% RSLogix 500 project MULTI_POSITION_SERVO.RSS, saved by version 8.30.00.16 %
PROJECT "UNTITLED"    % processor: Bul.1763 MicroLogix 1100 Series B %

PROGRAM FILES
  LAD 2 "MAIN"  4 rungs
  LAD 3 "I/O"  8 rungs
  LAD 4 "CONTROLS"  22 rungs

DATA FILES
  O0 OUTPUT  5 elements
  I1 INPUT  7 elements
  S2 STATUS  66 elements
  B3 BINARY  3 elements
  T4 TIMER  3 elements
  C5 COUNTER  1 elements
  R6 CONTROL  1 elements
  N7 INTEGER  2 elements
  F8 FLOAT  1 elements

LADDER 2 "MAIN"
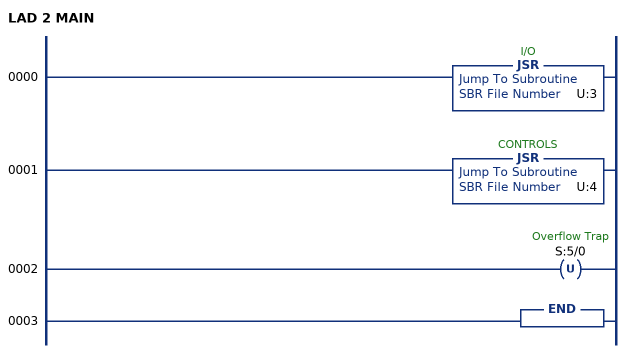
% Rung: 0 %
SOR JSR U:3 EOR
%   U:3  "I/O" %
% Rung: 1 %
SOR JSR U:4 EOR
%   U:4  "CONTROLS" %
% Rung: 2 %
SOR OTU S:5/0 EOR
%   S:5/0  "Overflow Trap" %
% Rung: 3 %
SOR END EOR

LADDER 3 "I/O"
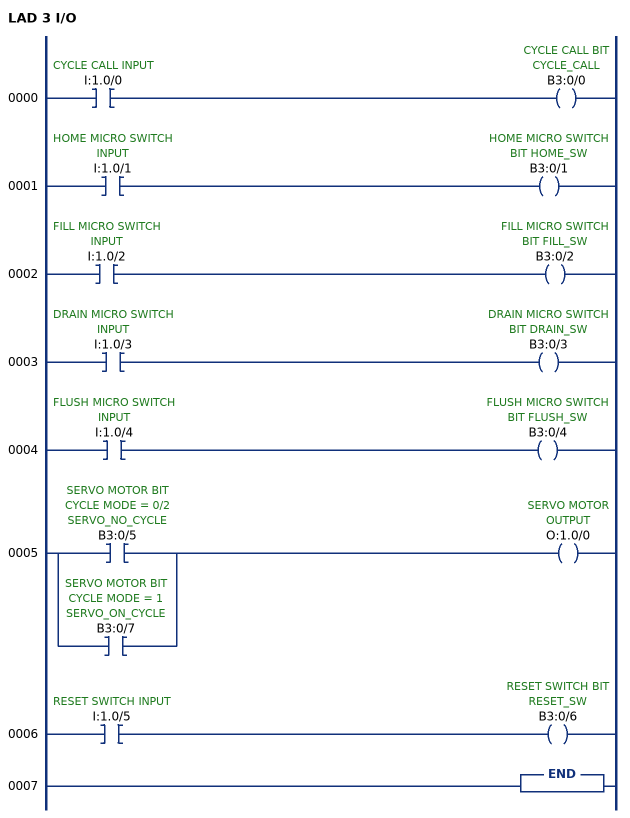
% Rung: 0 %
SOR XIC I:1.0/0 OTE B3:0/0 EOR
%   I:1.0/0  "CYCLE CALL INPUT" %
%   B3:0/0  CYCLE_CALL  "CYCLE CALL BIT" %
% Rung: 1 %
SOR XIC I:1.0/1 OTE B3:0/1 EOR
%   I:1.0/1  "HOME MICRO SWITCH INPUT" %
%   B3:0/1  HOME_SW  "HOME MICRO SWITCH BIT" %
% Rung: 2 %
SOR XIC I:1.0/2 OTE B3:0/2 EOR
%   I:1.0/2  "FILL MICRO SWITCH INPUT" %
%   B3:0/2  FILL_SW  "FILL MICRO SWITCH BIT" %
% Rung: 3 %
SOR XIC I:1.0/3 OTE B3:0/3 EOR
%   I:1.0/3  "DRAIN MICRO SWITCH INPUT" %
%   B3:0/3  DRAIN_SW  "DRAIN MICRO SWITCH BIT" %
% Rung: 4 %
SOR XIC I:1.0/4 OTE B3:0/4 EOR
%   I:1.0/4  "FLUSH MICRO SWITCH INPUT" %
%   B3:0/4  FLUSH_SW  "FLUSH MICRO SWITCH BIT" %
% Rung: 5 %
SOR BST XIC B3:0/5 NXB XIC B3:0/7 BND OTE O:1.0/0 EOR
%   B3:0/5  SERVO_NO_CYCLE  "SERVO MOTOR BIT CYCLE MODE = 0/2" %
%   B3:0/7  SERVO_ON_CYCLE  "SERVO MOTOR BIT CYCLE MODE = 1" %
%   O:1.0/0  "SERVO MOTOR OUTPUT" %
% Rung: 6 %
SOR XIC I:1.0/5 OTE B3:0/6 EOR
%   I:1.0/5  "RESET SWITCH INPUT" %
%   B3:0/6  RESET_SW  "RESET SWITCH BIT" %
% Rung: 7 %
SOR END EOR

LADDER 4 "CONTROLS"
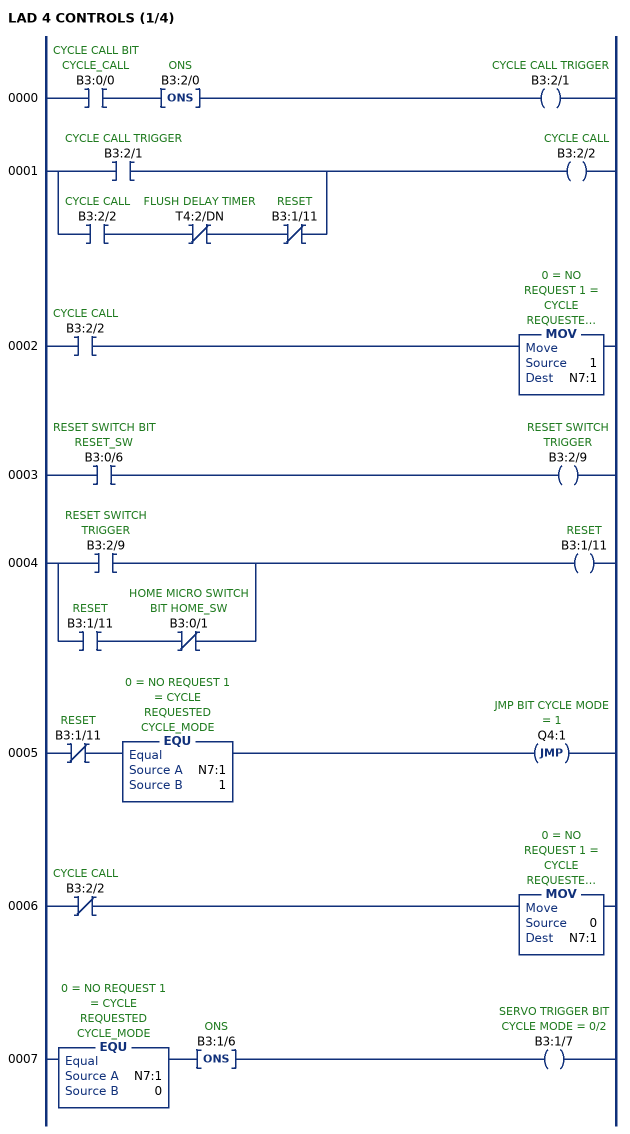
% Rung: 0 %
SOR XIC B3:0/0 ONS B3:2/0 OTE B3:2/1 EOR
%   B3:0/0  CYCLE_CALL  "CYCLE CALL BIT" %
%   B3:2/0  "ONS" %
%   B3:2/1  "CYCLE CALL TRIGGER" %
% Rung: 1 %
SOR BST XIC B3:2/1 NXB XIC B3:2/2 XIO T4:2/DN XIO B3:1/11 BND OTE B3:2/2 EOR
%   B3:2/1  "CYCLE CALL TRIGGER" %
%   B3:2/2  "CYCLE CALL" %
%   T4:2/DN  "FLUSH DELAY TIMER" %
%   B3:1/11  "RESET" %
% Rung: 2 %
SOR XIC B3:2/2 MOV 1 N7:1 EOR
%   B3:2/2  "CYCLE CALL" %
%   N7:1  CYCLE_MODE  "0 = NO REQUEST 1 = CYCLE REQUESTED" %
% Rung: 3 %
SOR XIC B3:0/6 OTE B3:2/9 EOR
%   B3:0/6  RESET_SW  "RESET SWITCH BIT" %
%   B3:2/9  "RESET SWITCH TRIGGER" %
% Rung: 4 %
SOR BST XIC B3:2/9 NXB XIC B3:1/11 XIO B3:0/1 BND OTE B3:1/11 EOR
%   B3:2/9  "RESET SWITCH TRIGGER" %
%   B3:1/11  "RESET" %
%   B3:0/1  HOME_SW  "HOME MICRO SWITCH BIT" %
% Rung: 5 %
SOR XIO B3:1/11 EQU N7:1 1 JMP Q4:1 EOR
%   B3:1/11  "RESET" %
%   N7:1  CYCLE_MODE  "0 = NO REQUEST 1 = CYCLE REQUESTED" %
%   Q4:1  "JMP BIT CYCLE MODE = 1" %
% Rung: 6 %
SOR XIO B3:2/2 MOV 0 N7:1 EOR
%   B3:2/2  "CYCLE CALL" %
%   N7:1  CYCLE_MODE  "0 = NO REQUEST 1 = CYCLE REQUESTED" %
% Rung: 7 %
SOR EQU N7:1 0 ONS B3:1/6 OTE B3:1/7 EOR
%   N7:1  CYCLE_MODE  "0 = NO REQUEST 1 = CYCLE REQUESTED" %
%   B3:1/6  "ONS" %
%   B3:1/7  "SERVO TRIGGER BIT CYCLE MODE = 0/2" %

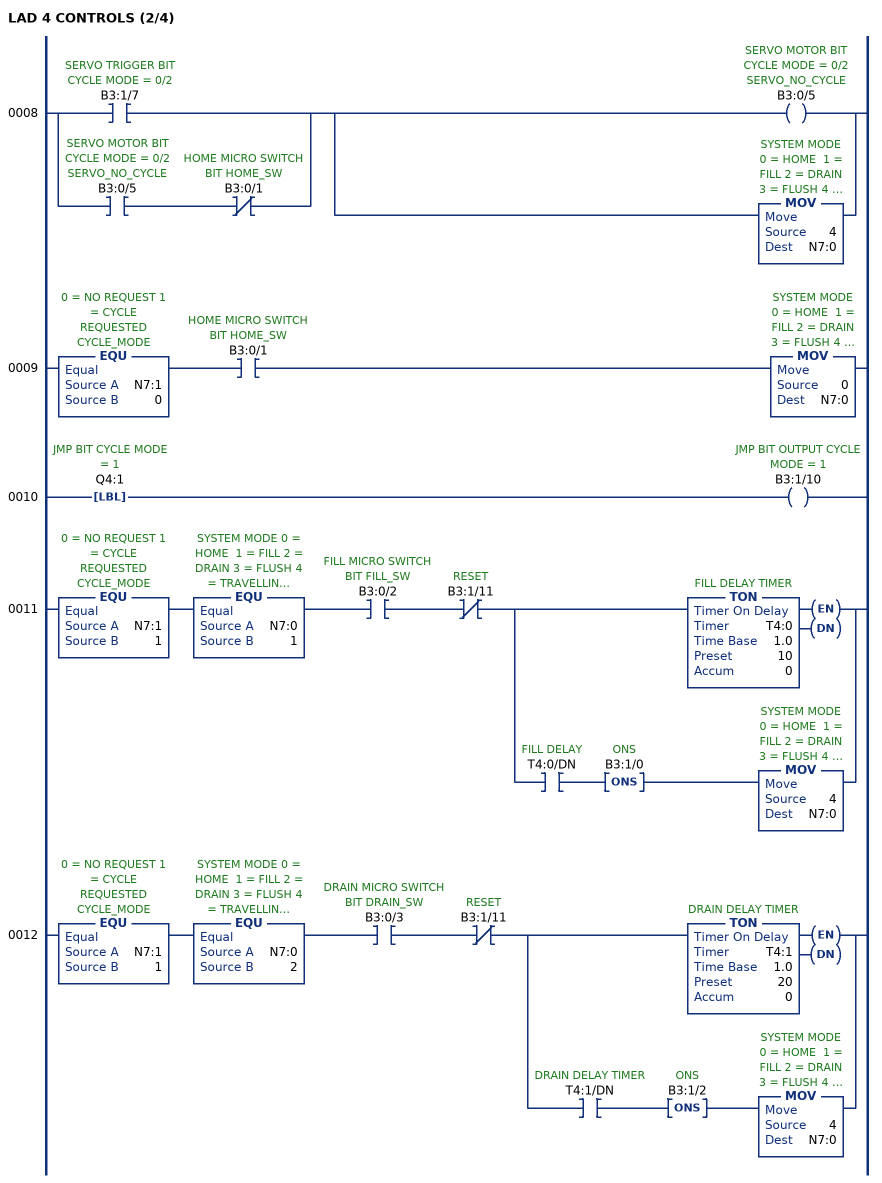
% Rung: 8 %
SOR BST XIC B3:1/7 NXB XIC B3:0/5 XIO B3:0/1 BND BST OTE B3:0/5 NXB MOV 4 N7:0 BND EOR
%   B3:1/7  "SERVO TRIGGER BIT CYCLE MODE = 0/2" %
%   B3:0/5  SERVO_NO_CYCLE  "SERVO MOTOR BIT CYCLE MODE = 0/2" %
%   B3:0/1  HOME_SW  "HOME MICRO SWITCH BIT" %
%   N7:0  SYSTEM_MODE  "SYSTEM MODE 0 = HOME  1 = FILL 2 = DRAIN 3 = FLUSH 4 = TRAVELLING" %
% Rung: 9 %
SOR EQU N7:1 0 XIC B3:0/1 MOV 0 N7:0 EOR
%   N7:1  CYCLE_MODE  "0 = NO REQUEST 1 = CYCLE REQUESTED" %
%   B3:0/1  HOME_SW  "HOME MICRO SWITCH BIT" %
%   N7:0  SYSTEM_MODE  "SYSTEM MODE 0 = HOME  1 = FILL 2 = DRAIN 3 = FLUSH 4 = TRAVELLING" %
% Rung: 10 %
SOR LBL Q4:1 OTE B3:1/10 EOR
%   Q4:1  "JMP BIT CYCLE MODE = 1" %
%   B3:1/10  "JMP BIT OUTPUT CYCLE MODE = 1" %
% Rung: 11 %
SOR EQU N7:1 1 EQU N7:0 1 XIC B3:0/2 XIO B3:1/11 BST TON T4:0 1.0 10 0 NXB XIC T4:0/DN ONS B3:1/0 MOV 4 N7:0 BND EOR
%   N7:1  CYCLE_MODE  "0 = NO REQUEST 1 = CYCLE REQUESTED" %
%   N7:0  SYSTEM_MODE  "SYSTEM MODE 0 = HOME  1 = FILL 2 = DRAIN 3 = FLUSH 4 = TRAVELLING" %
%   B3:0/2  FILL_SW  "FILL MICRO SWITCH BIT" %
%   B3:1/11  "RESET" %
%   T4:0  "FILL DELAY TIMER" %
%   T4:0/DN  "FILL DELAY" %
%   B3:1/0  "ONS" %
% Rung: 12 %
SOR EQU N7:1 1 EQU N7:0 2 XIC B3:0/3 XIO B3:1/11 BST TON T4:1 1.0 20 0 NXB XIC T4:1/DN ONS B3:1/2 MOV 4 N7:0 BND EOR
%   N7:1  CYCLE_MODE  "0 = NO REQUEST 1 = CYCLE REQUESTED" %
%   N7:0  SYSTEM_MODE  "SYSTEM MODE 0 = HOME  1 = FILL 2 = DRAIN 3 = FLUSH 4 = TRAVELLING" %
%   B3:0/3  DRAIN_SW  "DRAIN MICRO SWITCH BIT" %
%   B3:1/11  "RESET" %
%   T4:1  "DRAIN DELAY TIMER" %
%   T4:1/DN  "DRAIN DELAY TIMER" %
%   B3:1/2  "ONS" %

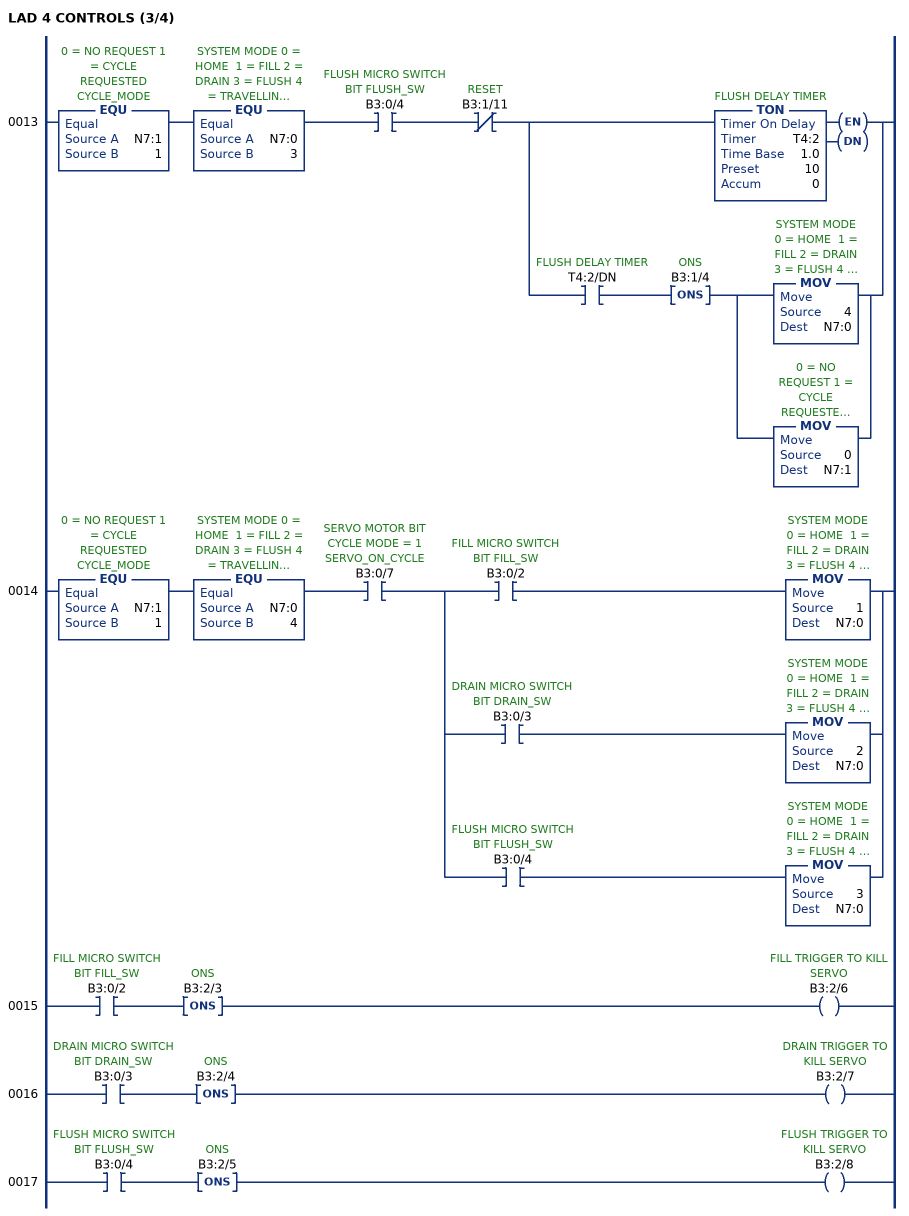
% Rung: 13 %
SOR EQU N7:1 1 EQU N7:0 3 XIC B3:0/4 XIO B3:1/11 BST TON T4:2 1.0 10 0 NXB XIC T4:2/DN ONS B3:1/4 BST MOV 4 N7:0 NXB MOV 0 N7:1 BND BND EOR
%   N7:1  CYCLE_MODE  "0 = NO REQUEST 1 = CYCLE REQUESTED" %
%   N7:0  SYSTEM_MODE  "SYSTEM MODE 0 = HOME  1 = FILL 2 = DRAIN 3 = FLUSH 4 = TRAVELLING" %
%   B3:0/4  FLUSH_SW  "FLUSH MICRO SWITCH BIT" %
%   B3:1/11  "RESET" %
%   T4:2  "FLUSH DELAY TIMER" %
%   T4:2/DN  "FLUSH DELAY TIMER" %
%   B3:1/4  "ONS" %
% Rung: 14 %
SOR EQU N7:1 1 EQU N7:0 4 XIC B3:0/7 BST XIC B3:0/2 MOV 1 N7:0 NXB XIC B3:0/3 MOV 2 N7:0 NXB XIC B3:0/4 MOV 3 N7:0 BND EOR
%   N7:1  CYCLE_MODE  "0 = NO REQUEST 1 = CYCLE REQUESTED" %
%   N7:0  SYSTEM_MODE  "SYSTEM MODE 0 = HOME  1 = FILL 2 = DRAIN 3 = FLUSH 4 = TRAVELLING" %
%   B3:0/7  SERVO_ON_CYCLE  "SERVO MOTOR BIT CYCLE MODE = 1" %
%   B3:0/2  FILL_SW  "FILL MICRO SWITCH BIT" %
%   B3:0/3  DRAIN_SW  "DRAIN MICRO SWITCH BIT" %
%   B3:0/4  FLUSH_SW  "FLUSH MICRO SWITCH BIT" %
% Rung: 15 %
SOR XIC B3:0/2 ONS B3:2/3 OTE B3:2/6 EOR
%   B3:0/2  FILL_SW  "FILL MICRO SWITCH BIT" %
%   B3:2/3  "ONS" %
%   B3:2/6  "FILL TRIGGER TO KILL SERVO" %
% Rung: 16 %
SOR XIC B3:0/3 ONS B3:2/4 OTE B3:2/7 EOR
%   B3:0/3  DRAIN_SW  "DRAIN MICRO SWITCH BIT" %
%   B3:2/4  "ONS" %
%   B3:2/7  "DRAIN TRIGGER TO KILL SERVO" %
% Rung: 17 %
SOR XIC B3:0/4 ONS B3:2/5 OTE B3:2/8 EOR
%   B3:0/4  FLUSH_SW  "FLUSH MICRO SWITCH BIT" %
%   B3:2/5  "ONS" %
%   B3:2/8  "FLUSH TRIGGER TO KILL SERVO" %

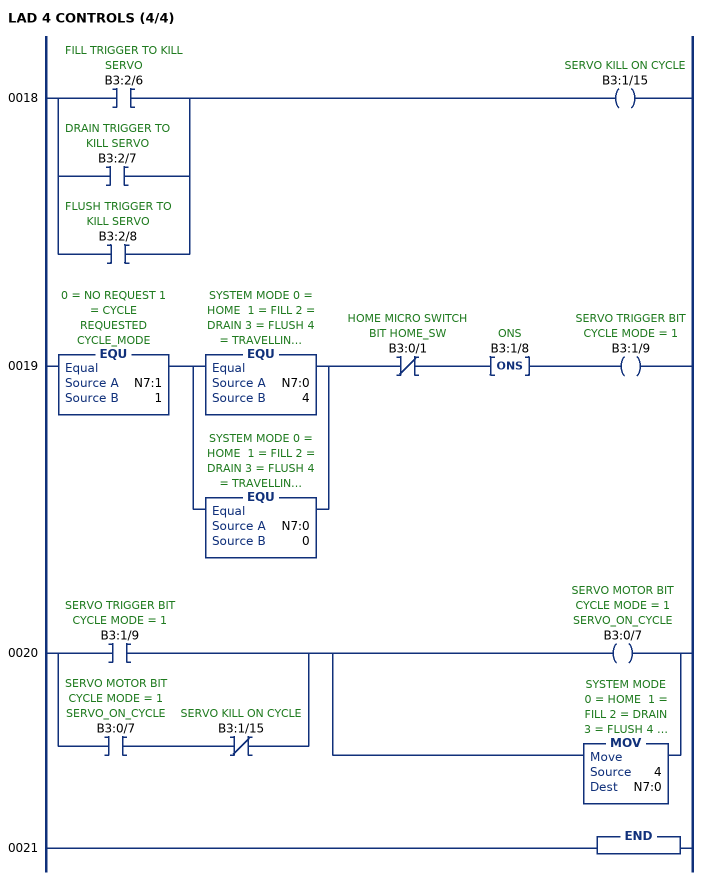
% Rung: 18 %
SOR BST XIC B3:2/6 NXB XIC B3:2/7 NXB XIC B3:2/8 BND OTE B3:1/15 EOR
%   B3:2/6  "FILL TRIGGER TO KILL SERVO" %
%   B3:2/7  "DRAIN TRIGGER TO KILL SERVO" %
%   B3:2/8  "FLUSH TRIGGER TO KILL SERVO" %
%   B3:1/15  "SERVO KILL ON CYCLE" %
% Rung: 19 %
SOR EQU N7:1 1 BST EQU N7:0 4 NXB EQU N7:0 0 BND XIO B3:0/1 ONS B3:1/8 OTE B3:1/9 EOR
%   N7:1  CYCLE_MODE  "0 = NO REQUEST 1 = CYCLE REQUESTED" %
%   N7:0  SYSTEM_MODE  "SYSTEM MODE 0 = HOME  1 = FILL 2 = DRAIN 3 = FLUSH 4 = TRAVELLING" %
%   B3:0/1  HOME_SW  "HOME MICRO SWITCH BIT" %
%   B3:1/8  "ONS" %
%   B3:1/9  "SERVO TRIGGER BIT CYCLE MODE = 1" %
% Rung: 20 %
SOR BST XIC B3:1/9 NXB XIC B3:0/7 XIO B3:1/15 BND BST OTE B3:0/7 NXB MOV 4 N7:0 BND EOR
%   B3:1/9  "SERVO TRIGGER BIT CYCLE MODE = 1" %
%   B3:0/7  SERVO_ON_CYCLE  "SERVO MOTOR BIT CYCLE MODE = 1" %
%   B3:1/15  "SERVO KILL ON CYCLE" %
%   N7:0  SYSTEM_MODE  "SYSTEM MODE 0 = HOME  1 = FILL 2 = DRAIN 3 = FLUSH 4 = TRAVELLING" %
% Rung: 21 %
SOR END EOR

OTHER DOCUMENTED ADDRESSES
  B3:1/1  "DRAIN MODE TRIGGER BIT"
  B3:1/3  "FLUSH CYCLE TRIGGER BIT"
  B3:1/5  "CYCLE END TRIGGER"
  B3:1/12  "FILL TRIGGER BIT"
  B3:1/13  "DRAIN TRIGGER BIT"
  B3:1/14  "FLUSH TRIGGER BIT"
  I:0  "CYCLE CALL"
  I:0.0/0  "CYCLE CALL INPUT"

DATA TABLE (non-zero values as saved)
DATA T4
% .PRE .ACC %
% T4:0 % 10 0
% T4:1 % 20 0
% T4:2 % 10 0
